FUNCTION_BLOCK FB_FieldCodecBool IMPLEMENTS I_FieldCodec
VAR_INPUT
END_VAR
VAR_OUTPUT
END_VAR
VAR
    bValue : BOOL;
END_VAR

METHOD CalculatePackedDataSize : HRESULT
VAR_INPUT CONSTANT
	anyFirstElem	: T_Any;
	nLength	        : UDINT;        // items to write
END_VAR
VAR_OUTPUT
    nPackedDataSize : UDINT;
END_VAR
VAR
    anyItem         : T_ANY;
    i               : UDINT;
    nValue          : BYTE;
END_VAR
anyItem := anyFirstElem;

IF nLength < 1 THEN
    nPackedDataSize := 0;
    RETURN;
END_IF

FOR i := 0  TO nLength - 1 DO
    anyItem.pValue := anyFirstElem.pValue + (i * TO_UDINT(anyFirstElem.diSize)); 
    nValue := PBYTE_TO_BYTE(anyItem.pValue);
    nPackedDataSize := nPackedDataSize + GCL_PB.cBoolSize;
END_FOR
END_METHOD

{warning 'Add property implementation'}
(* Gets the end tag of the codec or 0 if there is no end tag*)
PROPERTY EndTag : UDINT
GET
END_GET
END_PROPERTY

{warning 'Add property implementation'}
PROPERTY ipMessage : I_Message
GET
END_GET
SET
END_SET
END_PROPERTY

METHOD IsPackedRepeatedField : BOOL
VAR_INPUT
	nTag	: UDINT;
END_VAR
IsPackedRepeatedField := F_IsPackedRepeatedField(nTag);
END_METHOD

{warning 'Add property implementation'}
PROPERTY pParseContext : POINTER TO FB_ParseContext
SET
END_SET
END_PROPERTY

{warning 'Add property implementation'}
PROPERTY pWriteContext : POINTER TO FB_WriteContext
SET
END_SET
END_PROPERTY

{warning 'Add property implementation'}
(* Gets the tag of the codec.*)
PROPERTY Tag : UDINT
GET
END_GET
END_PROPERTY


METHOD ValueReader : HRESULT
VAR_IN_OUT
    stCtx : ST_ParseContext;
END_VAR
VAR_OUTPUT
	anyOut	: T_Any;
END_VAR

ValueReader := F_ParseRawVarint32(stCtx, bValue);
anyOut := F_ToAnyType(anyArg:= bValue);
END_METHOD

METHOD ValueWriter : HRESULT
VAR_IN_OUT
    stCtx  : ST_WriteContext;
END_VAR
VAR_INPUT
    anyIn : T_ANY;
END_VAR
VAR
	nValue : BYTE;
END_VAR

nValue := PBYTE_TO_BYTE(anyIn.pValue);
ValueWriter := F_WriteRawByte(stCtx, nValue);
END_METHOD

END_FUNCTION_BLOCK

(* stored: Version 1.1.0.1
   POU FB_FieldCodecBool: Id {3214d183-fb88-47d2-976d-5db1da0bbb6f}, SpecialFunc None
   Method CalculatePackedDataSize: Id {a59e0abc-6ed9-4fdb-9d25-08792bfaeff4}
   Property EndTag: Id {b0652fba-7df5-4545-8c7f-0850470ca4cd}
   Get Get: Id {bb89d1d9-b315-44f7-bb1c-57d9f08efb17}
   Property ipMessage: Id {0531ec29-8b53-4761-b3a4-2da48b8006cc}
   Get Get: Id {710498bf-02e2-41e3-b026-4ad385c77bf5}
   Set Set: Id {72b8bcf8-ca41-463e-80cf-e95201647657}
   Method IsPackedRepeatedField: Id {126ed474-6ba0-475d-a48c-511e198d9b17}
   Property pParseContext: Id {795b2c22-46bb-4731-b2ca-5642eea669be}
   Set Set: Id {5fb8fdef-8ad4-43fa-8b58-9a8446c02e7b}
   Property pWriteContext: Id {cd4df9ea-9490-4676-862c-77adba5b1e66}
   Set Set: Id {10e2074d-97f7-4c5d-bf76-81987da15aeb}
   Property Tag: Id {eed3c457-8418-46c9-8f34-1d7647661c60}
   Get Get: Id {4eea2bf2-8a03-4538-9b3e-31aeab368569}
   Method ValueReader: Id {6e4d75e5-f6e6-42d1-8e60-72d496f7021f}
   Method ValueWriter: Id {5fa0bf78-e845-4e96-96fd-c3bc2aa1bcd5} *)
